FUNCTION_BLOCK Outlet_EStop EXTENDS Outlet_State IMPLEMENTS I_Call
VAR
	_bCanDeactivate	: BOOL;
END_VAR

METHOD Call
VAR_INPUT
	iTag	: Broadcast.Tags.I_Tag;
END_VAR
IF _ctx.smgr.Current = _ctx.iEStop THEN
	IF iTag.Option = 'UNSAFE' THEN
		_bCanDeactivate := TRUE;
		_ctx.smgr.Request(_ctx.iOperational);
	END_IF
ELSE
	IF iTag.Option = 'SAFE' THEN
		_bCanDeactivate := FALSE;
		_ctx.smgr.Request(_ctx.iEStop);
	END_IF
END_IF
END_METHOD

METHOD CanDeactivate : BOOL
CanDeactivate := _bCanDeactivate;
END_METHOD

METHOD OnInit
_ctx.bDrainValveOpen := FALSE;
END_METHOD

END_FUNCTION_BLOCK

(* stored: Version 1.1.0.1
   POU Outlet_EStop: Id {be40cdf2-e169-405c-b44c-e53f7aa9401c}, SpecialFunc None
   Method Call: Id {d89dcd10-be3c-4290-b890-5d803ea2de06}
   Method CanDeactivate: Id {87eff437-f586-46fe-b483-26fd89d2c643}
   Method OnInit: Id {9da3af7c-9d5b-428f-bd23-f29e2a47405e} *)
